PROGRAM Buffer_IMU
VAR
	pSec		: WORD;
	diff		: BOOL;
	
	TimeStr		: ARRAY [1..50] OF STRING;
	//Millis		: ARRAY [1..50] OF STRING;
	Trailer_ID_Lead	: ARRAY [1..50] OF STRING;
	//RoadSec		: ARRAY [1..50] OF STRING;
	Pitch_Lead		: ARRAY [1..50] OF STRING;
	Roll_Lead		: ARRAY [1..50] OF STRING;
	AccX_Lead		: ARRAY [1..50] OF STRING;
	AccY_Lead		: ARRAY [1..50] OF STRING;
	AccZ_Lead		: ARRAY [1..50] OF STRING;
	
	Trailer_ID_Rear	: ARRAY [1..50] OF STRING;
	//RoadSec		: ARRAY [1..50] OF STRING;
	Pitch_Rear		: ARRAY [1..50] OF STRING;
	Roll_Rear		: ARRAY [1..50] OF STRING;
	AccX_Rear		: ARRAY [1..50] OF STRING;
	AccY_Rear		: ARRAY [1..50] OF STRING;
	AccZ_Rear		: ARRAY [1..50] OF STRING;
	
	fbSqlDatabase	: FB_SQLDatabaseEvt(sNetID := '', tTimeout := T#1000S);
	fbSqlCommand	: FB_SQLCommandEvt(sNetID := '', tTimeout := T#1000S);
	fbSqlResult		: FB_SQLResultEvt(sNetID:='', tTimeout   := T#1000S); 
	sCmd			: STRING(500000);
	sCmd2			: STRING(500000);
	nState			: INT;
	nState_Switch	: INT;
	
	aReadStruct		: ST_SelectStructIMU;
	aReadStruct_2	: ST_SelectStructIMU;
	Timestamp		: DT;
	Timestamp_2		: DT; 
	
	Initialized		: BOOL := FALSE;
	Done			: BOOL;
	i				: INT;
	Pragma_Done		: BOOL;
	Counter			: ULINT;
	
	Dbid			: UDINT;
	
	bDisconnect		: BOOL;
END_VAR

(* convert to strings *)
//PrimeMover_ID		:= Read_ID.PrimeMover_ID;
TimeStr				:= Read_IMU.TimeStr;
//Millis			:= Read_IMU.Millis;
Trailer_ID_Lead		:= Read_IMU.Trailer_ID_Lead;
Pitch_Lead			:= Read_IMU.Pitch_Lead;
Roll_Lead			:= Read_IMU.Roll_Lead;
AccX_Lead			:= Read_IMU.AccX_Lead;
AccY_Lead			:= Read_IMU.AccY_Lead;
AccZ_Lead			:= Read_IMU.AccZ_Lead;

Trailer_ID_Rear		:= Read_IMU.Trailer_ID_Rear;
Pitch_Rear			:= Read_IMU.Pitch_Rear;
Roll_Rear			:= Read_IMU.Roll_Rear;
AccX_Rear			:= Read_IMU.AccX_Rear;
AccY_Rear			:= Read_IMU.AccY_Rear;
AccZ_Rear			:= Read_IMU.AccZ_Rear;

IF NOT Initialized THEN
	
	//initialization (choose which database for buffer)
	CASE nState OF
				
		0:
			(* connect to buffer_imu *)	
			IF Vacuum_Buffer_IMU.Vacuumed THEN
				
				Dbid := 2;		
				IF fbSqlDatabase.Connect(Dbid) THEN
					IF fbSqlDatabase.bError THEN
						nState := 255; 
					ELSE
						nState := nState+1;
					END_IF
				END_IF
				
			END_IF
			
			
		1:
			IF fbSqlDatabase.CreateCmd(ADR(fbSqlCommand)) THEN
				IF fbSqlDatabase.bError THEN
					nState := 255; 
				ELSE
					nState := nState+1; 
				END_IF
			END_IF
			
		2:	(* execute pragmas *)
			sCmd	:= 'PRAGMA journal_mode = WAL; PRAGMA synchronous = NORMAL; PRAGMA temp_store = MEMORY; PRAGMA mmap_size = 30000000000; PRAGMA page_size = 32768; PRAGMA locking_mode = EXCLUSIVE;';
			
			IF fbSQLCommand.Execute(ADR(sCmd), SIZEOF(sCmd)) THEN
				IF fbSQLCommand.bError THEN
					nState := 255; 
				ELSE
					nState := nState+1; 
				END_IF
			END_IF
			
		3:
			(* select oldest data from buffer_imu *)
			sCmd	:= 'SELECT * FROM `buffer_imu` ORDER BY datetime ASC LIMIT 1';
			
			IF fbSQLCommand.ExecuteDataReturn(ADR(sCmd), SIZEOF(sCmd), ADR(fbSqlResult)) THEN
				IF fbSQLCommand.bError THEN
					nState := 255; 
				ELSE
					nState := nState+1; 
				END_IF
			END_IF
			
		4:
			IF fbSqlResult.Read(0, 1, ADR(aReadStruct), SIZEOF(aReadStruct), TRUE, TRUE) THEN
				IF fbSqlResult.bError THEN
					nState := 255; 
				ELSE
					nState := nState+1; 
				END_IF
			END_IF
			
		5:
			IF fbSqlResult.Release() THEN
				IF fbSqlResult.bError THEN
					nState := 255;
				ELSE
					nState := nState+1;
				END_IF
			END_IF
			
		6:	(* execute pragma optimize *)
			sCmd	:= 'PRAGMA optimize;';
			
			IF fbSQLCommand.Execute(ADR(sCmd), SIZEOF(sCmd)) THEN
				IF fbSQLCommand.bError THEN
					nState := 255; 
				ELSE
					nState := nState+1; 
				END_IF
			END_IF
			
		7:
			(* disconnect from buffer_imu *)
			IF fbSqlDatabase.Disconnect() THEN
				IF fbSqlDatabase.bError THEN
					nState := 255;
				ELSE
					nState := nState+1;
				END_IF
			END_IF
			
		8:	
			(* connect to buffer_imu_2 *)
			IF Vacuum_Buffer_IMU_2.Vacuumed THEN
				
				Dbid := 5;	
				IF fbSqlDatabase.Connect(Dbid) THEN
					IF fbSqlDatabase.bError THEN
						nState := 255; 
					ELSE
						nState := nState+1;
					END_IF
				END_IF
				
			END_IF	
			
		9:
			IF fbSqlDatabase.CreateCmd(ADR(fbSqlCommand)) THEN
				IF fbSqlDatabase.bError THEN
					nState := 255; 
				ELSE
					nState := nState+1; 
				END_IF
			END_IF
			
		10:	(* execute pragmas *)
			sCmd	:= 'PRAGMA journal_mode = WAL; PRAGMA synchronous = NORMAL; PRAGMA temp_store = MEMORY; PRAGMA mmap_size = 30000000000; PRAGMA page_size = 32768; PRAGMA locking_mode = EXCLUSIVE;';
			
			IF fbSQLCommand.Execute(ADR(sCmd), SIZEOF(sCmd)) THEN
				IF fbSQLCommand.bError THEN
					nState := 255; 
				ELSE
					nState := nState+1; 
				END_IF
			END_IF
			
		11:
			(* select oldest data from buffer_imu *)
			sCmd	:= 'SELECT * FROM `buffer_imu` ORDER BY datetime ASC LIMIT 1';
			
			IF fbSQLCommand.ExecuteDataReturn(ADR(sCmd), SIZEOF(sCmd), ADR(fbSqlResult)) THEN
				IF fbSQLCommand.bError THEN
					nState := 255; 
				ELSE
					nState := nState+1; 
				END_IF
			END_IF
			
		12:
			IF fbSqlResult.Read(0, 1, ADR(aReadStruct_2), SIZEOF(aReadStruct_2), TRUE, TRUE) THEN
				IF fbSqlResult.bError THEN
					nState := 255; 
				ELSE
					nState := nState+1; 
				END_IF
			END_IF
			
		13:
			IF fbSqlResult.Release() THEN
				IF fbSqlResult.bError THEN
					nState := 255;
				ELSE
					nState := nState+1;
				END_IF
			END_IF
			
		14:	(* execute pragma optimize *)
			sCmd	:= 'PRAGMA optimize;';
			
			IF fbSQLCommand.Execute(ADR(sCmd), SIZEOF(sCmd)) THEN
				IF fbSQLCommand.bError THEN
					nState := 255; 
				ELSE
					nState := nState+1; 
				END_IF
			END_IF
			
		15:
			(* disconnect from buffer_imu_2 *)
			IF bDisconnect := fbSqlDatabase.Disconnect() THEN
				IF fbSqlDatabase.bError THEN
					nState := 255;
				ELSE
					nState := nState+1;
				END_IF
			END_IF
			
		16:
			// compare oldest data
			aReadStruct.datetime 	:= REPLACE(aReadStruct.datetime, '-', 1, 11);
			aReadStruct_2.datetime 	:= REPLACE(aReadStruct_2.datetime, '-', 1, 11);
			
			Timestamp	:= SYSTEMTIME_TO_DT(STRING_TO_SYSTEMTIME(aReadStruct.datetime));
			Timestamp_2	:= SYSTEMTIME_TO_DT(STRING_TO_SYSTEMTIME(aReadStruct_2.datetime));

			IF Timestamp = DT#1970-1-1-00:00:00 THEN
				Dbid := 2;
			ELSIF Timestamp_2 = DT#1970-1-1-00:00:00 THEN
				Dbid := 5;
			ELSIF Timestamp > Timestamp_2 THEN
				Dbid := 2;
			ELSE
				Dbid := 5;
			END_IF
			
			Initialized := TRUE;
			nState		:= 0;
			
		255:
			nState := 0;
			
	END_CASE

ELSE	
	
	(* save data to buffer every second *)
	IF diff:= Background_Time.cSec <> pSec THEN
		
		//database switching
		IF Get_IMU.Switch AND Counter >= 250 THEN
			
			CASE nState_Switch OF
				
				0:	(* execute pragma optimize *)
					sCmd	:= 'PRAGMA optimize;';
					
					IF fbSQLCommand.Execute(ADR(sCmd), SIZEOF(sCmd)) THEN
						IF fbSQLCommand.bError THEN
							nState_Switch := 255; 
						ELSE
							nState_Switch := nState_Switch+1; 
						END_IF
					END_IF
				
				1:
					IF fbSqlDatabase.bConnected THEN
						fbSqlDatabase.Disconnect();
					ELSE
						IF Dbid = 2 THEN
							Dbid := 5;
						ELSE
							Dbid := 2;
						END_IF
						Counter			:= 0;
						nState_Switch 	:= 0;
						Pragma_Done		:= FALSE;
					END_IF
					
				255:
					nState_Switch := 0;
					
			END_CASE
		
		ELSE
			
			IF Done THEN
				Done	:= FALSE;
				IF fbSqlDatabase.bConnected THEN
					nState 	:= 1;
				ELSE
					nState 	:= 0;
				END_IF	
			END_IF
			
			CASE nState OF	
				0:	
					IF fbSqlDatabase.Connect(Dbid) THEN
						IF fbSqlDatabase.bError THEN
							nState := 255;
						ELSE
							nState := nState + 1; 
						END_IF
					END_IF
				
				1:
					IF fbSqlDatabase.CreateCmd(ADR(fbSqlCommand)) THEN
						IF fbSqlDatabase.bError THEN
							nState := 255; 
						ELSE
							nState := nState+1; 
						END_IF
					END_IF
					
				2:	(* execute pragmas *)
					IF NOT Pragma_Done THEN
						sCmd	:= 'PRAGMA journal_mode = WAL; PRAGMA synchronous = NORMAL; PRAGMA temp_store = MEMORY; PRAGMA mmap_size = 30000000000; PRAGMA page_size = 32768; PRAGMA locking_mode = EXCLUSIVE;';
					
						IF fbSQLCommand.Execute(ADR(sCmd), SIZEOF(sCmd)) THEN
							IF fbSQLCommand.bError THEN
								nState := 255; 
							ELSE
								nState 		:= nState+1; 
								Pragma_Done := TRUE;
							END_IF
						END_IF
					
					ELSE
						nState 		:= nState+1;
 
					END_IF
					
				3:	
					(* build query *)	
					sCmd:= 'INSERT INTO buffer_imu (datetime,trailer_id_lead,trailer_id_rear,pitch_lead,roll_lead,ax_lead,ay_lead,az_lead,pitch_rear,roll_rear,ax_rear,ay_rear,az_rear) VALUES ';
					
					FOR i := 1 TO 50 BY 1 DO
						sCmd2:= CONCAT('($'', TimeStr[i]);
						sCmd2:= CONCAT(sCmd2, '$',');
						sCmd2:= CONCAT(sCmd2, Trailer_ID_Lead[i]);
						sCmd2:= CONCAT(sCmd2, ',');
						sCmd2:= CONCAT(sCmd2, Trailer_ID_Rear[i]);
						sCmd2:= CONCAT(sCmd2, ',');
						sCmd2:= CONCAT(sCmd2, Pitch_Lead[i]);
						sCmd2:= CONCAT(sCmd2, ',');
						sCmd2:= CONCAT(sCmd2, Roll_Lead[i]);
						sCmd2:= CONCAT(sCmd2, ',');
						sCmd2:= CONCAT(sCmd2, AccX_Lead[i]);
						sCmd2:= CONCAT(sCmd2, ',');
						sCmd2:= CONCAT(sCmd2, AccY_Lead[i]);
						sCmd2:= CONCAT(sCmd2, ',');
						sCmd2:= CONCAT(sCmd2, AccZ_Lead[i]);
						sCmd2:= CONCAT(sCmd2, ',');
						sCmd2:= CONCAT(sCmd2, Pitch_Rear[i]);
						sCmd2:= CONCAT(sCmd2, ',');
						sCmd2:= CONCAT(sCmd2, Roll_Rear[i]);
						sCmd2:= CONCAT(sCmd2, ',');
						sCmd2:= CONCAT(sCmd2, AccX_Rear[i]);
						sCmd2:= CONCAT(sCmd2, ',');
						sCmd2:= CONCAT(sCmd2, AccY_Rear[i]);
						sCmd2:= CONCAT(sCmd2, ',');
						sCmd2:= CONCAT(sCmd2, AccZ_Rear[i]);
						
						IF i = 50 THEN
							sCmd2:= CONCAT(sCmd2, ')');
						ELSE	
							sCmd2:= CONCAT(sCmd2, '),');
						END_IF
						
						CONCAT2(ADR(sCmd), ADR(sCmd2), ADR(sCmd), SIZEOF(sCmd));
					END_FOR
					
					
					IF fbSQLCommand.Execute(ADR(sCmd), SIZEOF(sCmd)) THEN
						IF fbSQLCommand.bError THEN
							nState := 255; 
						ELSE
							nState := nState+1; 
							pSec := Background_Time.cSec;
							
						END_IF
					END_IF
					
				4: 
					Counter := Counter + 50;
					Done	:= TRUE;
						
				255:
					nState := 0;
					
			END_CASE	
			
		END_IF
	END_IF
END_IF

END_PROGRAM

(* stored: Version 1.1.0.1, ProductVersion 3.1.4024.6
   POU Buffer_IMU: Id {5645648d-eb13-4929-86df-ef282757094e}, SpecialFunc None *)
